DATA_BLOCK "DebugData"
{ S7_Optimized_Access := "TRUE" }
VERSION: 0.1
NON_RETAIN
    VAR
        source { ExternalAccessible := 'False'; ExternalVisible := 'False'; ExternalWritable := 'False'} : Int;
        flag : Bool;
    END_VAR

BEGIN
    source := 1;

END_DATA_BLOCK

